INTERFACE ITF_HMIEMenu EXTENDS ITF_BaseControlElement

END_INTERFACE

(* stored: Version 1.1.0.1
   Itf ITF_HMIEMenu: Id {dc3b9d3c-c21c-4086-8483-fad3245993b2} *)
